// TIA Portal V17 export
// export: Created 2024-06-16T17:47:39.6165286Z, ExportSetting WithDefaults, DisplayName Totally Integrated Automation Portal, DisplayVersion V17, DisplayName TIA Portal Openness, DisplayVersion V17, DisplayName TIA Portal Version Control Interface, DisplayVersion V17, DisplayName STEP 7 Professional, DisplayVersion V17, DisplayName STEP 7 Safety, DisplayVersion V17, DisplayName WinCC Professional, DisplayVersion V17
VAR_GLOBAL   // PLC tag table "St3_In"
   IO_TrappeEntree_Ouvert AT %I2.4 : Bool;   // Trappe d'entrée : Ouverte
   IO_TrappeEntree_Fermee AT %I2.5 : Bool;   // Trappe d'entrée : Fermée
   IO_TrappeSortie_Ouvert AT %I2.6 : Bool;   // Trappe de sortie : Ouverte
   IO_TrappeSortie_Fermee AT %I2.7 : Bool;   // Trappe de sortie : Fermée
   IO_Obturateur_Ouvert AT %I3.0 : Bool;   // Obturateur : Ouvert
   IO_Obturateur_Fermee AT %I3.1 : Bool;   // Obturateur : Fermé
   IO_PorteRX_Ouvert AT %I3.2 : Bool;   // Porte RX : Ouverte (Homme)
   IO_PorteRX_Fermee AT %I3.3 : Bool;   // Porte RX : Ferméee (Homme)
   IO_Cpt_RX1 AT %I3.4 : Bool;   // Présence barquette en début de RX : RX1
   IO_Cpt_RX2 AT %I3.5 : Bool;   // Détection butée à came : RX2
   IO_Cpt_RX3 AT %I3.6 : Bool;   // Détection butée pivot : RX3
   IO_Vy_Orange AT %I3.7 : Bool;   // Obturateur Fermée + RX Actif
   IO_Vy_Rouge AT %I4.0 : Bool;   // Obturateur Ouvert + RX Actif
END_VAR
